// TIA Portal V19 export
VAR_GLOBAL   // PLC tag table "KP8"
   Jog_Reverse_Green_KP8 AT %Q51.5 : Bool;   // KP8
   Enable_Disable_KP8 AT %I50.7 : Bool;   // KP8
   Drive_Start_KP8 AT %I50.6 : Bool;   // KP8
   Jog_Reverse_KP8 AT %I50.5 : Bool;   // KP8
   Switch1_KP8 AT %I50.4 : Bool;   // KP8
   Enable_Disable_Green_KP8 AT %Q51.7 : Bool;   // KP8
   Drive_Start_Red_KP8 AT %Q50.6 : Bool;   // KP8
   Jog_Reverse_Red_KP8 AT %Q50.5 : Bool;   // KP8
   Switch1_Red_KP8 AT %Q50.4 : Bool;   // KP8
   RESET_KP8 AT %I50.3 : Bool;   // KP8
   Drive_Stop_KP8 AT %I50.2 : Bool;   // KP8
   Jog_Forward_KP8 AT %I50.1 : Bool;   // KP8
   RESET_Red_KP8 AT %Q50.3 : Bool;   // KP8
   Drive_Stop_Red_KP8 AT %Q50.2 : Bool;   // KP8
   Jog_Forward_Red_KP8 AT %Q50.1 : Bool;   // KP8
   Switch2_KP8 AT %I50.0 : Bool;   // KP8
   Switch2_Red_KP8 AT %Q50.0 : Bool;   // KP8
   Enable_Disable_Red_KP8 AT %Q50.7 : Bool;   // KP8
   Drive_Start_Green_KP8 AT %Q51.6 : Bool;   // KP8
   Switch1_Green_KP8 AT %Q51.4 : Bool;   // KP8
   RESET_Green_KP8 AT %Q51.3 : Bool;   // KP8
   Drive_Stop_Green_KP8 AT %Q51.2 : Bool;   // KP8
   Jog_Forward_Green_KP8 AT %Q51.1 : Bool;   // KP8
   Switch2_Green_KP8 AT %Q51.0 : Bool;   // KP8
   Switch2_Blue_KP8 AT %Q52.0 : Bool;   // KP8
   Jog_Forward_Blue_KP8 AT %Q52.1 : Bool;   // KP8
   Drive_Stop_Blue_KP8 AT %Q52.2 : Bool;   // KP8
   RESET_Blue_KP8 AT %Q52.3 : Bool;   // KP8
   Switch1_Blue_KP8 AT %Q52.4 : Bool;   // KP8
   Jog_Reverse_Blue_KP8 AT %Q52.5 : Bool;   // KP8
   Drive_Start_Blue_KP8 AT %Q52.6 : Bool;   // KP8
   Enable_Disable_Blue_KP8 AT %Q52.7 : Bool;   // KP8
   KP8_Red AT %QB50 : Byte;   // KP8
   KP8_Green AT %QB51 : Byte;   // KP8
   KP8_Blue AT %QB52 : Byte;   // KP8
END_VAR
